TYPE U_GEAR_DATA :
UNION
  stData              : ARRAY[1..MAX_MOVER] OF ST_GEAR_DATA;

  byData    AT %I*    : ARRAY[1..MAX_MOVER] OF
                        ARRAY[1..SIZEOF(ST_GEAR_DATA)] OF BYTE;
END_UNION
END_TYPE

(* stored: Version 1.1.0.1, ProductVersion 3.1.4026.13
   DUT U_GEAR_DATA: Id {24b4700d-189d-400c-9a09-b4267845b958} *)
